// TIA Portal project "Projeto Automação Industrial" (V15.1)
// Vorlageprojekt für das Buch mit Zielsystem S7-1200

(* hardware
DEVICE "S7-1200-Station_1"  S7-1200 Station
   slot 0: "Baugruppenträger_0"  Rack  V1.0
   slot 1: "PLC_1"  CPU 1211C DC/DC/DC  6ES7 211-1AE40-0XB0  V4.1
*)

// ===== PLC "PLC_1"  CPU 1211C DC/DC/DC =====

VAR_GLOBAL   // PLC tag table "Standard-Variablentabelle"
   "Liga esteira de entrada" AT %A0.0 : Bool;
   "Peça na saída da esteira de entrada" AT %E0.0 : Bool;
   "Botão Start" AT %E0.1 : Bool;
   "Luz indicadora - Botão Start" AT %Q1.1 : Bool;
   "Selo de funcionamento" AT %Q3.0 : Bool;
   "Peça azul detectada" AT %Q2.1 : Bool;
   "Peça verde detectada" AT %Q2.2 : Bool;
   "Peça cinza/metal detectada" AT %Q2.3 : Bool;
   "Lâmina de parada" AT %Q0.1 : Bool;
   "Virar ordenador 1" AT %Q0.3 : Bool;
   "Liga estaira - ordenador 1" AT %Q0.4 : Bool;
   "Parar esteira de entrada" AT %Q2.4 : Bool;
   "Sensor de visão" AT %ID30 : DInt;
   "Contador 1 - peças azuis" AT %QD30 : DInt;
   "Botão Stop" AT %I0.3 : Bool;
   "Saída do contador 1" AT %Q2.5 : Bool;
   "Timer de parada da esteira de entrada" AT %Q2.6 : Bool;
   "Contador 2 - peças verdes" AT %QD34 : DInt;
   "Saída do contador 2" AT %Q2.7 : Bool;
   "Contador 3 - peças cinza/metal" AT %QD38 : DInt;
   "Saída contador 3" AT %Q1.4 : Bool;
   "Liga esteira de saída" AT %Q0.2 : Bool;
   "Virar ordenador 2" AT %Q0.5 : Bool;
   "Liga estaira - ordenador 2" AT %Q0.6 : Bool;
   "Virar ordenador 3" AT %Q0.7 : Bool;
   "Liga esteira - ordenador 3" AT %Q1.0 : Bool;
   "Luz indicadora - Botão Stop" AT %Q1.3 : Bool;
   "Envio de peça concluído" AT %Q3.1 : Bool;
   "Timer de saída" AT %Q3.2 : Bool;
   "Botão Reset" AT %I0.2 : Bool;
   "Luz indicadora - Botão Reset" AT %Q1.2 : Bool;
END_VAR

// folder: System blocks/Program resources

DATA_BLOCK "IEC_Counter_0_DB"   // DB1
{ S7_Optimized_Access := 'TRUE' }
AUTHOR : Simatic
FAMILY : IEC
NAME : CNTR
VERSION : 1.0
// stored: InstanceOfName IEC_COUNTER
"IEC_COUNTER"
BEGIN
END_DATA_BLOCK

DATA_BLOCK "IEC_Timer_0_DB_4"   // DB3
{ S7_Optimized_Access := 'TRUE' }
AUTHOR : Simatic
FAMILY : IEC
NAME : IEC_TMR
VERSION : 1.0
// stored: InstanceOfName IEC_TIMER
"IEC_TIMER"
BEGIN
END_DATA_BLOCK

DATA_BLOCK "IEC_Counter_0_DB_1"   // DB5
{ S7_Optimized_Access := 'TRUE' }
AUTHOR : Simatic
FAMILY : IEC
NAME : CNTR
VERSION : 1.0
// stored: InstanceOfName IEC_COUNTER
"IEC_COUNTER"
BEGIN
END_DATA_BLOCK

DATA_BLOCK "IEC_Counter_0_DB_2"   // DB6
{ S7_Optimized_Access := 'TRUE' }
AUTHOR : Simatic
FAMILY : IEC
NAME : CNTR
VERSION : 1.0
// stored: InstanceOfName IEC_COUNTER
"IEC_COUNTER"
BEGIN
END_DATA_BLOCK

DATA_BLOCK "IEC_Timer_0_DB_3"   // DB9
{ S7_Optimized_Access := 'TRUE' }
AUTHOR : Simatic
FAMILY : IEC
NAME : IEC_TMR
VERSION : 1.0
// stored: InstanceOfName IEC_TIMER
"IEC_TIMER"
BEGIN
END_DATA_BLOCK

// folder: (top level)

FUNCTION "MHJ-PLC-Lab-Function-S71200" : Void   // FC9000, SCL
{ S7_Optimized_Access := 'TRUE' }
VERSION : 0.1
   VAR_TEMP
      rdTimeReturn : Int;
      outputTime : DTL;
      SyncVal : Byte;
      forVal : Int;
      forVal_2 : Int;
      Value : Byte;
   END_VAR
   VAR CONSTANT
      CompVal : Byte := 16#34;
      Value_01 : Byte := 16#11;
      Value_01_DW : DWord := 16#A165_D992;
      Value_02_DW : DWord := 16#58BE_4401;
   END_VAR
BEGIN

   #Value:=PEEK(area := 16#82,
        dbNumber := 0,
        byteOffset := 511);
   #Value := #Value + 1;

   POKE(area := 16#82,
        dbNumber := 0,
        byteOffset := 511,
        value := #Value);

   POKE(area:=16#81,
        dbNumber:=0,
        byteOffset:=1016,
        value:=#Value_01_DW);
   POKE(area := 16#81,
        dbNumber := 0,
        byteOffset := 1020,
        value := #Value_02_DW);

   POKE(area := 16#81,
        dbNumber := 0,
        byteOffset := 511,
        value := B#16#00);

   FOR #forVal := 0 TO 120 DO
       FOR #forVal_2:=0 TO 10 DO
           #rdTimeReturn:=RD_SYS_T(#outputTime);
           #rdTimeReturn := WR_SYS_T(#outputTime);
           #rdTimeReturn := RD_SYS_T(#outputTime);
           #rdTimeReturn := WR_SYS_T(#outputTime);
       END_FOR;
       #SyncVal:= PEEK(area := 16#81,
                      dbNumber := 0,
                      byteOffset := 511);
       IF #SyncVal = #CompVal THEN
          GOTO M_1;
       END_IF;
   END_FOR;
   RETURN;

   M_1:
   POKE(area := 16#81,
        dbNumber := 0,
        byteOffset := 511,
        value := B#16#0);
END_FUNCTION

ORGANIZATION_BLOCK "Main"   // OB1, LAD, ProgramCycle
TITLE = "Main Program Sweep (Cycle)"
{ S7_Optimized_Access := 'TRUE' }
VERSION : 0.1
   VAR_INPUT
      Initial_Call : Bool;   // Initial call of this OB
      Remanence : Bool;   // =True, if remanent data are available
   END_VAR
BEGIN

REGION Network 1: Konnektierungsbaustein für PLC-Lab / Biblioteca do CLP
   // Im Netzwerk 1 wird der Konnektierungsbaustein für PLC-Lab aufgerufen.
   // Dieser Aufruf darf nicht entfernt werden!
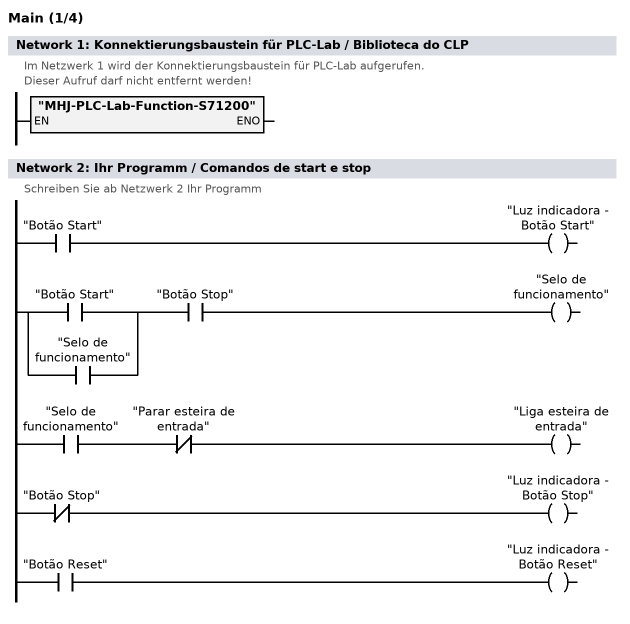
   RUNG wire#powerrail
      "MHJ-PLC-Lab-Function-S71200"()
   END_RUNG
   // the same network as SCL:
   "MHJ-PLC-Lab-Function-S71200"();
END_REGION

REGION Network 2: Ihr Programm / Comandos de start e stop
   // Schreiben Sie ab Netzwerk 2 Ihr Programm
   RUNG wire#powerrail
      Contact( "Botão Start" )
      Coil( "Luz indicadora - Botão Start" )
   END_RUNG
   RUNG wire#powerrail
      Contact( "Botão Start" )
      wire#w1
      Contact( "Botão Stop" )
      Coil( "Selo de funcionamento" )
   END_RUNG
   RUNG wire#powerrail
      Contact( "Selo de funcionamento" )
   END_RUNG wire#w1
   RUNG wire#powerrail
      Contact( "Selo de funcionamento" )
      I_Contact( "Parar esteira de entrada" )
      Coil( "Liga esteira de entrada" )
   END_RUNG
   RUNG wire#powerrail
      I_Contact( "Botão Stop" )
      Coil( "Luz indicadora - Botão Stop" )
   END_RUNG
   RUNG wire#powerrail
      Contact( "Botão Reset" )
      Coil( "Luz indicadora - Botão Reset" )
   END_RUNG
   // the same network as SCL:
   "Luz indicadora - Botão Start" := "Botão Start";
   "Selo de funcionamento" := ("Botão Start" OR "Selo de funcionamento") AND "Botão Stop";
   "Liga esteira de entrada" := "Selo de funcionamento" AND NOT "Parar esteira de entrada";
   "Luz indicadora - Botão Stop" := NOT "Botão Stop";
   "Luz indicadora - Botão Reset" := "Botão Reset";
END_REGION

REGION Network 3: Lógica do sensor de visão
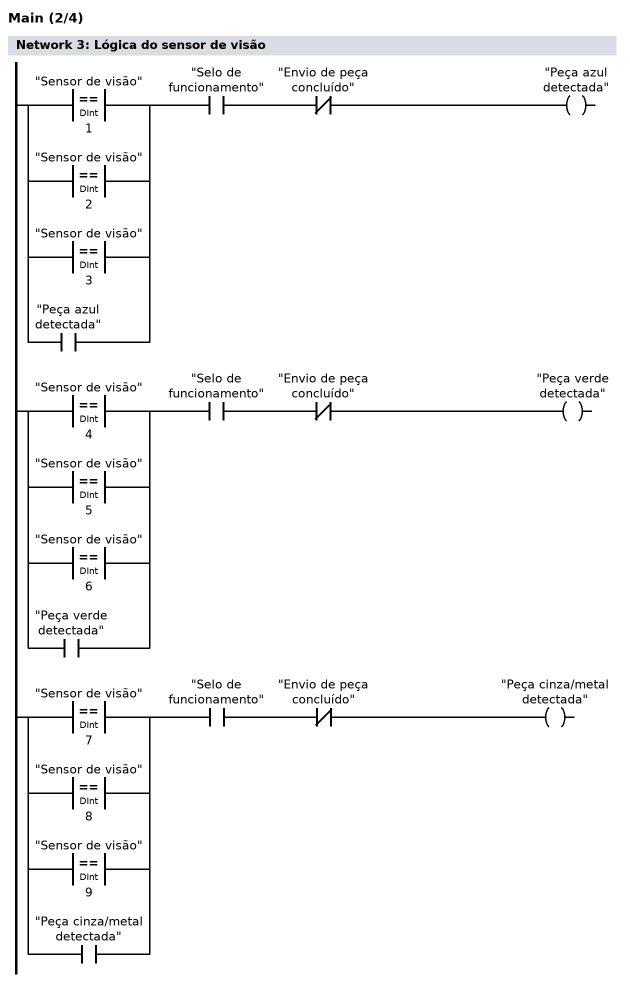
   RUNG wire#powerrail
      { S7_Templates := "SrcType := DInt" } EQ_Contact(in1 := "Sensor de visão", in2 := 1)
      wire#w1
      Contact( "Selo de funcionamento" )
      I_Contact( "Envio de peça concluído" )
      Coil( "Peça azul detectada" )
   END_RUNG
   RUNG wire#powerrail
      { S7_Templates := "SrcType := DInt" } EQ_Contact(in1 := "Sensor de visão", in2 := 2)
   END_RUNG wire#w1
   RUNG wire#powerrail
      { S7_Templates := "SrcType := DInt" } EQ_Contact(in1 := "Sensor de visão", in2 := 3)
   END_RUNG wire#w1
   RUNG wire#powerrail
      Contact( "Peça azul detectada" )
   END_RUNG wire#w1
   RUNG wire#powerrail
      { S7_Templates := "SrcType := DInt" } EQ_Contact(in1 := "Sensor de visão", in2 := 4)
      wire#w2
      Contact( "Selo de funcionamento" )
      I_Contact( "Envio de peça concluído" )
      Coil( "Peça verde detectada" )
   END_RUNG
   RUNG wire#powerrail
      { S7_Templates := "SrcType := DInt" } EQ_Contact(in1 := "Sensor de visão", in2 := 5)
   END_RUNG wire#w2
   RUNG wire#powerrail
      { S7_Templates := "SrcType := DInt" } EQ_Contact(in1 := "Sensor de visão", in2 := 6)
   END_RUNG wire#w2
   RUNG wire#powerrail
      Contact( "Peça verde detectada" )
   END_RUNG wire#w2
   RUNG wire#powerrail
      { S7_Templates := "SrcType := DInt" } EQ_Contact(in1 := "Sensor de visão", in2 := 7)
      wire#w3
      Contact( "Selo de funcionamento" )
      I_Contact( "Envio de peça concluído" )
      Coil( "Peça cinza/metal detectada" )
   END_RUNG
   RUNG wire#powerrail
      { S7_Templates := "SrcType := DInt" } EQ_Contact(in1 := "Sensor de visão", in2 := 8)
   END_RUNG wire#w3
   RUNG wire#powerrail
      { S7_Templates := "SrcType := DInt" } EQ_Contact(in1 := "Sensor de visão", in2 := 9)
   END_RUNG wire#w3
   RUNG wire#powerrail
      Contact( "Peça cinza/metal detectada" )
   END_RUNG wire#w3
   // the same network as SCL:
   "Peça azul detectada" := (("Sensor de visão" = 1) OR ("Sensor de visão" = 2) OR ("Sensor de visão" = 3) OR "Peça azul detectada") AND "Selo de funcionamento" AND NOT "Envio de peça concluído";
   "Peça verde detectada" := (("Sensor de visão" = 4) OR ("Sensor de visão" = 5) OR ("Sensor de visão" = 6) OR "Peça verde detectada") AND "Selo de funcionamento" AND NOT "Envio de peça concluído";
   "Peça cinza/metal detectada" := (("Sensor de visão" = 7) OR ("Sensor de visão" = 8) OR ("Sensor de visão" = 9) OR "Peça cinza/metal detectada") AND "Selo de funcionamento" AND NOT "Envio de peça concluído";
END_REGION

REGION Network 4: Lógica dos ordenadores
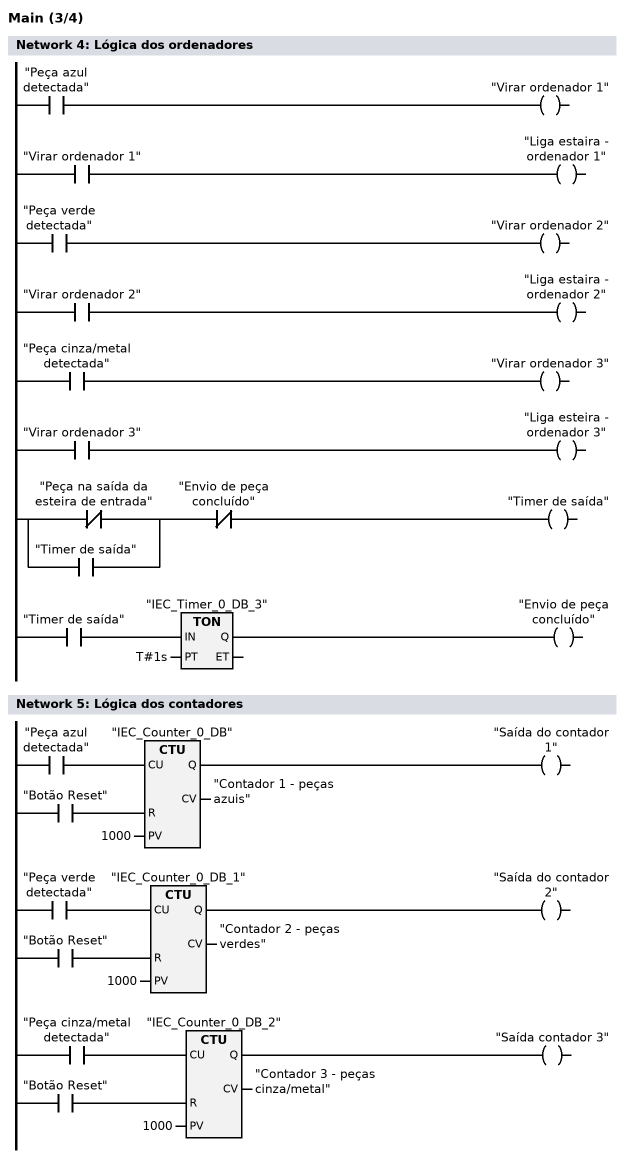
   "Virar ordenador 1" := "Peça azul detectada";
   "Liga estaira - ordenador 1" := "Virar ordenador 1";
   "Virar ordenador 2" := "Peça verde detectada";
   "Liga estaira - ordenador 2" := "Virar ordenador 2";
   "Virar ordenador 3" := "Peça cinza/metal detectada";
   "Liga esteira - ordenador 3" := "Virar ordenador 3";
   "Timer de saída" := (NOT "Peça na saída da esteira de entrada" OR "Timer de saída") AND NOT "Envio de peça concluído";
   "IEC_Timer_0_DB_3".TON(IN := "Timer de saída", PT := T#1s);
   "Envio de peça concluído" := "IEC_Timer_0_DB_3".Q;
END_REGION

REGION Network 5: Lógica dos contadores
   "IEC_Counter_0_DB".CTU(CU := "Peça azul detectada",
                          R := "Botão Reset",
                          PV := 1000,
                          CV => "Contador 1 - peças azuis");
   "Saída do contador 1" := "IEC_Counter_0_DB".Q;
   "IEC_Counter_0_DB_1".CTU(CU := "Peça verde detectada",
                           R := "Botão Reset",
                           PV := 1000,
                           CV => "Contador 2 - peças verdes");
   "Saída do contador 2" := "IEC_Counter_0_DB_1".Q;
   "IEC_Counter_0_DB_2".CTU(CU := "Peça cinza/metal detectada",
                           R := "Botão Reset",
                           PV := 1000,
                           CV => "Contador 3 - peças cinza/metal");
   "Saída contador 3" := "IEC_Counter_0_DB_2".Q;
END_REGION

REGION Network 6: Lógica de parada da esteira de entrada
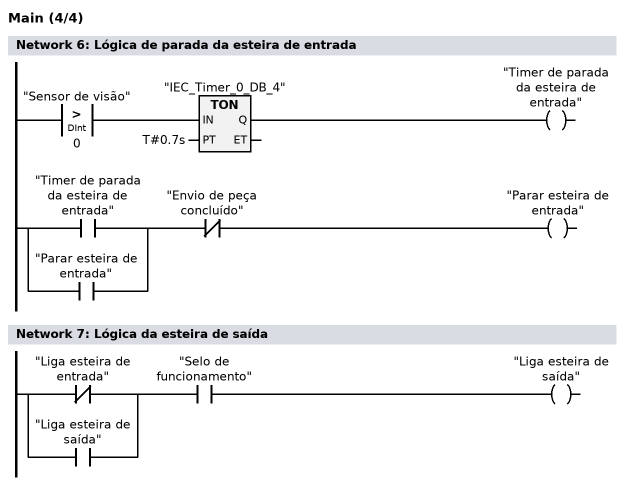
   "IEC_Timer_0_DB_4".TON(IN := "Sensor de visão" > 0, PT := T#0.7s);
   "Timer de parada da esteira de entrada" := "IEC_Timer_0_DB_4".Q;
   "Parar esteira de entrada" := ("Timer de parada da esteira de entrada" OR "Parar esteira de entrada") AND NOT "Envio de peça concluído";
END_REGION

REGION Network 7: Lógica da esteira de saída
   RUNG wire#powerrail
      I_Contact( "Liga esteira de entrada" )
      wire#w1
      Contact( "Selo de funcionamento" )
      Coil( "Liga esteira de saída" )
   END_RUNG
   RUNG wire#powerrail
      Contact( "Liga esteira de saída" )
   END_RUNG wire#w1
   // the same network as SCL:
   "Liga esteira de saída" := (NOT "Liga esteira de entrada" OR "Liga esteira de saída") AND "Selo de funcionamento";
END_REGION
END_ORGANIZATION_BLOCK